TYPE dt_Parameters :
STRUCT
	Scale	: LREAL;
	Etc		: INT;
END_STRUCT
END_TYPE

(* stored: Version 1.1.0.1, ProductVersion 3.1.4024.15
   DUT dt_Parameters: Id {98217eab-4fbd-4168-978d-ef6b79e58c8e} *)
